TYPE ST_Modbus_WriteRequest :
STRUCT

	WriteRegVals: 					ARRAY[1..10] OF WORD;
	SlaveAddress : 					UINT;
	QtyWordsToWrite : 				UINT;
	AdrFirstSlaveRegisterWrite : 	UINT;
	bRequestCompleted: 				BOOL;
	bRequestAccepted: 				BOOL;

END_STRUCT
END_TYPE

(* stored: Version 1.1.0.1, ProductVersion 3.1.4024.12
   DUT ST_Modbus_WriteRequest: Id {ed34aa93-193d-4c86-97f1-12574307e791} *)
